{attribute 'no_check'}
//Returns a string found on the left side of a seperator, empty if seperator is not found
FUNCTION readStrToSeperator : T_MaxString
VAR_INPUT
	Seperator												:	STRING(10) :=';';
	Strline													:	T_MaxString;
END_VAR
VAR_IN_OUT
END_VAR
VAR
	pos														:	INT;
END_VAR

IF strline='' 
THEN
	readStrToSeperator										:= '';
ELSE
	pos 													:= FIND (strline,seperator);
	IF (pos >= 1) 
	THEN
		readStrToSeperator									:= LEFT (strline,pos-1);
	ELSE
		readStrToSeperator									:= '';
	END_IF
END_IF

END_FUNCTION

(* stored: Version 1.1.0.1, ProductVersion 3.1.4024.3
   POU readStrToSeperator: Id {351ca5e1-2b55-4d32-870e-61d70c7dcb63}, SpecialFunc None *)
